// SIMATIC S7-200 project (STEP 7-Micro/WIN), CPU 224 REL 02.00

ORGANIZATION_BLOCK MAIN:OB1
TITLE=PROGRAM COMMENTS
BEGIN
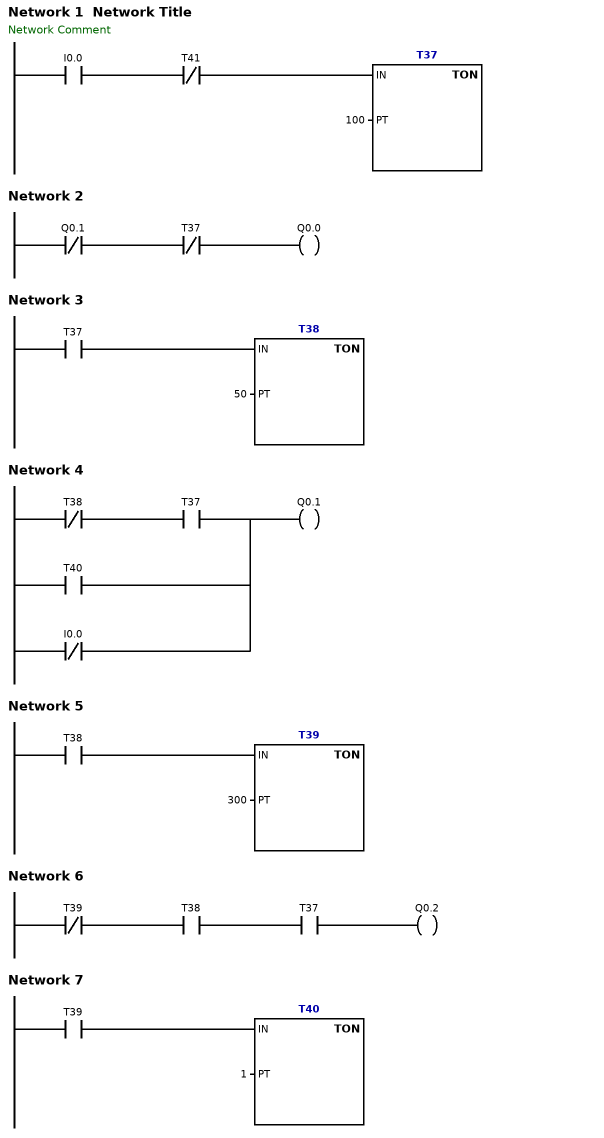
Network 1 // Network Title
// Network Comment
LD     I0.0
AN     T41
TON    T37, 100
Network 2
LDN    Q0.1
AN     T37
=      Q0.0
Network 3
LD     T37
TON    T38, 50
Network 4
LDN    T38
A      T37
O      T40
ON     I0.0
=      Q0.1
Network 5
LD     T38
TON    T39, 300
Network 6
LDN    T39
A      T38
A      T37
=      Q0.2
Network 7
LD     T39
TON    T40, 1
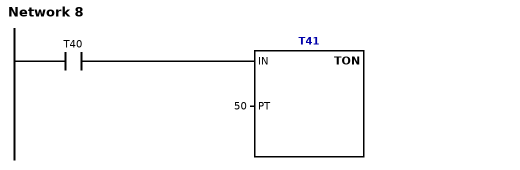
Network 8
LD     T40
TON    T41, 50
END_ORGANIZATION_BLOCK
